Staubli VAL3: selectAxis.pjx

--- selectAxis.pjx ---
Parameters version=s7.2.1 stackSize=5000 millimeterUnit=true
Program file=loadPage.pgx
Program file=main.pgx
Program file=onEnterEvent.pgx
Program file=onExit.pgx
Program file=onF1Event.pgx
Program file=onF2Event.pgx
Program file=onF3Event.pgx
Program file=onF4Event.pgx
Program file=onF5Event.pgx
Program file=onF6Event.pgx
Program file=onF7Event.pgx
Program file=onF8Event.pgx
Program file=onStart.pgx
Program file=refresh.pgx
Program file=refreshDynamic.pgx
Program file=refreshStatic.pgx
Data file=selectAxis.dtx
Library alias=use path=Disk://kernel/userPage/userPage.pjx
Library alias=io path=Disk://io/io.pjx
Library alias=page path=Disk://kernel/template/page/page.pjx
Library alias=language path=Disk://kernel/language/language.pjx

--- selectAxis.dtx ---
num nKey = -1
public num nPage = 10
num nRefresh = 498.406
num nTime = 1
num nValue[4]
  [0] = 1
  [1] = 2
  [2] = 3
  [3] = 4
string sDeeperSession
public string sItems
string sMenu[8]
  [0] = "Program Menu"
  [1] = "Trajectory Menu"
  [2] = "Enable laser"
  [3] = "Table frame"
  [4] = "PRODUCTION PAGE"
  [6] = "Advance"
  [7] = "Quit"
string sMenu8[8]
string sMessage
string sPathSession
string sSession
string sVersion = "ValTending 6.1.3.1"
bool bButton[8]
  [0] = true
  [1] = true
  [2] = true
  [3] = true
  [4] = true
  [6] = true
  [7] = true
bool bLaserOn
bool bInterlock

--- main.pgx ---
public program main()
  local bool l_bExit
begin
  // INIT
  //call onStart()
  // LOOP UNTIL Exit

  call refreshStatic()
  do
    // call the refresh
    call refresh()
    // take the key
    nKey=getKey()
    switch nKey
      case 271
        // select AXIS7
        call onF1Event()
      break
      case 272
        // select AXIS8
        call onF2Event()
      break
      case 273
        //
        call onF3Event()
      break
      case 274
        call onF4Event()
      break
      case 275
        //
        call onF5Event()
      break
      case 276
        //
        call onF6Event()
      break
      case 277
        //
        call onF7Event()
      break
      case 278
        //
        call onF8Event(l_bExit)
      break
      case 270
        call onEnterEvent()
      break
    endSwitch
    // release the resource
    delay(0)
  until nKey==255
  // on Exit
  //call onExit()
end

--- loadPage.pgx ---
program loadPage(string x_sPage, string& x_sItems[])
// load the next page
  local num i
  local string l_sMessage
  local num l_nClock
begin
  // look if the page libload is correct
  i=page:libLoad(x_sPage)
  if i!=0
    logMsg("[VALlaser] INTERFACE:PAGE LIBLOAD "+x_sPage+" result "+toString("",i))
    call language:message(l_sMessage,-7)
    popUpMsg(l_sMessage+x_sPage+" ; "+toString("",i))
  else
    // copy all the field from x_sItems to the next page
    call use:stringCopy(x_sItems,page:sItems)
    call page:main()
    // to give back
    call use:stringCopy(page:sItems,x_sItems)
  endIf
end

--- onEnterEvent.pgx ---
program onEnterEvent()
begin
end

--- onExit.pgx ---
program onExit()
begin
  //
  //  Kill everything
  logMsg("[VALlaser] INTERFACE:Quit")
  use:nToSuperV=1
  //
  //
end

--- onF1Event.pgx ---
program onF1Event()
  local num i
  local string l_sItem
begin
  // load the page AXIS7

end

--- onF2Event.pgx ---
program onF2Event()
  local string l_sItem
begin
 // look if the bButton is enable
  call loadPage("instrSequential/AXIS7/page_axis",l_sItem)
end

--- onF3Event.pgx ---
program onF3Event()
  local string l_sMessage
  local string l_sItem
begin

     // load the page AXIS8


end

--- onF4Event.pgx ---
program onF4Event()
  local num i
  local string l_sMessage
  local string l_sItem
begin
  // look if the bButton is enable
call loadPage("instrSequential/AXIS8/page_axis",l_sItem)
end

--- onF5Event.pgx ---
program onF5Event()
begin

end

--- onF6Event.pgx ---
program onF6Event()
  local string l_sItem
begin
  // look if the bButton is enable

end

--- onF7Event.pgx ---
program onF7Event()
  local num local1
begin
  // look if the bButton is enable

end

--- onF8Event.pgx ---
program onF8Event(bool& x_bExit[])
  local string l_sMessage
  local string l_sButton[2]
  local num l_nIndex
  local string l_sEvent
  local num l_nKey
begin
  // look if the bButton is enable

end

--- onStart.pgx ---
program onStart()
  local num i
begin
  // wait the START

end

--- refresh.pgx ---
program refresh()
// // page refresh
begin
  // refresh the static message
  if (nKey>=270 and nKey<=278) or use:bUseRefresh
    call refreshStatic()
    call refreshDynamic()
  else
    // refresh the Dynamic message
    if (clock()-nRefresh>nTime)
      call refreshDynamic()
    endIf
  endIf
  // release the resource
  delay(0)
end

--- refreshDynamic.pgx ---
program refreshDynamic()
begin
  // DO NOT CHANGE
  nRefresh=clock()
  //
  // ADD HERE
  //
  use:bUseRefresh=false
end

--- refreshStatic.pgx ---
program refreshStatic()
  local string l_sMessage[2]
  local string l_sMenu
  local string l_sSession
begin
  cls()
  //
  gotoxy(1,1)
  put("F2  AXIS7")
  gotoxy(1,3)
  put("F4  AXIS8")
  gotoxy(5,13)
  put("AXIS7")
  gotoxy(15,13)
  put("AXIS8")
  //
end
